{attribute addProperty BoxType "AT2026-0250-0019"}
{attribute addProperty Id "A_0077_AT2001_5250_0018_AT2001_5250AT2001_C5E5984862678.25"}
{attribute addProperty CRC "3813130644"}
{attribute addProperty SizeInBites "626"}
{attribute addProperty SizeInBytes "78.25"}
TYPE A_0065_AT2026_0250_0019_AT2026_0250_E347C194 EXTENDS AT2026_BA5A9548 :
STRUCT
	{attribute addProperty Name "A_0077_AT2001_5250_0018_AT2001_5250"}
	A_0077_AT2001_5250_0018_AT2001_5250 : AT2001_C5E59848;
END_STRUCT
END_TYPE

(* stored: Version 1.2.0.0, ProductVersion 3.1.4024.9
   DUT A_0065_AT2026_0250_0019_AT2026_0250_E347C194: Id {b37634fc-6ccd-4cd5-bbd9-e589f8e86d41} *)
